PROGRAM MAIN
VAR
	bVariableToLink  AT %I* : BOOL;
	
END_VAR

END_PROGRAM

(* stored: Version 1.1.0.1, ProductVersion 3.1.4024.10
   POU MAIN: Id {48bfe0e8-d73d-4fdd-873f-80e4de83eb30}, SpecialFunc None *)
